TYPE DUT_PARAMETER_OUTPUT :
STRUCT
	///Free to use = TRUE, busy to use =FALSE
	Dummy: BOOL := TRUE;
	///ID of the parameter
	ID: UINT;
	///Name of the parameter
	Name: STRING(80);
	///Unit of the parameter
	Unit: STRING(80);
	///Optional parameter
	Required: BOOL;
	///Default parameter to work
	Default: LREAL;
	///Minimum value of the parameter
	MinValue: LREAL;
	///Maximum value of the parameter
	MaxValue: LREAL;
END_STRUCT
END_TYPE

(* stored: Version 1.1.0.1, ProductVersion 3.1.0.25
   DUT DUT_PARAMETER_OUTPUT: Id {fa1d4e6f-8687-4ab8-84d2-82cc339f7ce0} *)
